PROGRAM IP237
VAR
	
	timer				: TON;
	nState				: INT := STATE_INIT;
	
	fbInit237_01_5500			: FB_InitPM;
	fbInit237_02_5500			: FB_InitPM;
	fbInit237_03_5500			: FB_InitPM;
	fbInit237_04_5500			: FB_InitPM;
	fbInit237_05_5500			: FB_InitPM;
	
	fbRead237_01_5500			: FB_PM_ION_9000;
	fbRead237_02_5500			: FB_PM_ION_9000;
	
	//Update 29-08-2022
	fbRead237_03_5500			: FB_ReadPM5350;
	
	//Update 29-08-2022
	fbRead237_04_5500			: FB_ReadPM5350;
	
	//Update 29-08-2022
	fbRead237_05_5500			: FB_ReadPM5350;
	
	
	ipAddr						: STRING := '10.91.37.237';
	nCount						: DINT;
	nQuantity					: WORD:=125;
	nMBAddr						: WORD:=1;
	bExec						: BOOL;
	bBusy						: BOOL;
	bError						: BOOL;
	nErrorId					:UDINT;
	cbRead						: UDINT;
	bOnTest						:bool;
	PMRawDataTest				:ST_PowerMeter;
	// UPDATE BY SUN
	fbInit237_06_5350			: FB_InitPM;
	fbInit237_07_5350			: FB_InitPM;
	fbInit237_08_5350			: FB_InitPM;
	fbInit237_09_5350			: FB_InitPM;
	fbInit237_10_5350			: FB_InitPM;
	fbInit237_11_5350			: FB_InitPM;
	fbInit237_12_5350			: FB_InitPM;
	fbInit237_13_5350			: FB_InitPM;
	
	fbRead237_06_5350			: FB_ReadPM5350;
	fbRead237_07_5350			: FB_ReadPM5350;
	fbRead237_08_5350			: FB_ReadPM5350;
	fbRead237_09_5350			: FB_ReadPM5350;
	fbRead237_10_5350			: FB_ReadPM5350;
	fbRead237_11_5350			: FB_ReadPM5350;
	fbRead237_12_5350			: FB_ReadPM5350;
	fbRead237_13_5350			: FB_ReadPM5350;
	
END_VAR

VAR CONSTANT
	STATE_INIT			:	INT		:= 0;
	STATE_WAIT_CMD		: 	INT		:= 5;
	STATE_READ1			:	INT		:= 10;
	STATE_READ2			:	INT		:= 20;
	STATE_READ3			:	INT		:= 30;
	STATE_READ4			:	INT		:= 40;
	STATE_READ5			:	INT		:= 50;
	////////////////////////////////////////
	STATE_READ6 		:	INT		:= 60;
	STATE_READ7			:	INT		:= 70;
	STATE_READ8			:	INT		:= 80;
	STATE_READ9			:	INT		:= 90;
	STATE_READ10		:	INT		:= 100;
	STATE_READ11		:	INT		:= 110;
	STATE_READ12		:	INT		:= 120;
	STATE_READ13		:	INT		:= 130;
		

END_VAR

CASE nState OF
	STATE_INIT:
		fbInit237_01_5500(	sIpAddress	:= '10.91.37.227',
							nPort		:= 502,
							nUnitID		:= 255,
							PM			:= pmDev.DB07_01_5500);
		fbInit237_02_5500(	sIpAddress	:= '10.91.37.228',
							nPort		:= 502,
							nUnitID		:= 255,
							PM			:= pmDev.DB07_02_5500);
		fbInit237_03_5500(	sIpAddress	:= '10.91.37.237',
							nPort		:= 502,
							nUnitID		:= 3,
							PM			:= pmDev.DB07_03_5500);
		fbInit237_04_5500(	sIpAddress	:= '10.91.37.237',
							nPort		:= 502,
							nUnitID		:= 4,
							PM			:= pmDev.DB07_04_5500);
		fbInit237_05_5500(	sIpAddress	:= '10.91.37.237',
							nPort		:= 502,
							nUnitID		:= 5,
							PM			:= pmDev.DB07_05_5500);
		// updata by sun///////////////////////////////////////////////
		
		fbInit237_06_5350(	sIpAddress	:= '10.91.37.237',
							nPort		:= 502,
							nUnitID		:= 6,
							PM			:= pmDev.DB07_06_5350);
							
		fbInit237_07_5350(	sIpAddress	:= '10.91.37.237',
							nPort		:= 502,
							nUnitID		:= 7,
							PM			:= pmDev.DB07_07_5350);
							
		fbInit237_08_5350(	sIpAddress	:= '10.91.37.237',
							nPort		:= 502,
							nUnitID		:= 8,
							PM			:= pmDev.DB07_08_5350);
							
		fbInit237_09_5350(	sIpAddress	:= '10.91.37.237',
							nPort		:= 502,
							nUnitID		:= 9,
							PM			:= pmDev.DB07_09_5350);
							
		fbInit237_10_5350(	sIpAddress	:= '10.91.37.237',
							nPort		:= 502,
							nUnitID		:= 10,
							PM			:= pmDev.DB07_10_5350);
							
		fbInit237_11_5350(	sIpAddress	:= '10.91.37.237',
							nPort		:= 502,
							nUnitID		:= 11,
							PM			:= pmDev.DB07_11_5350);
							
		fbInit237_12_5350(	sIpAddress	:= '10.91.37.237',
							nPort		:= 502,
							nUnitID		:= 12,
							PM			:= pmDev.DB07_12_5350);
							
		fbInit237_13_5350(	sIpAddress	:= '10.91.37.237',
							nPort		:= 502,
							nUnitID		:= 13,
							PM			:= pmDev.DB07_13_5350);
							
		timer(In:=TRUE, PT:= TIME_INIT);
		IF timer.Q THEN
			timer(In:=FALSE);
			nState	:= STATE_WAIT_CMD;
		END_IF
			
	STATE_WAIT_CMD:
			;
			
	STATE_READ1:
		fbRead237_01_5500(
			bExecute:=TRUE,
			PM:= pmDev.DB07_01_5500);
		IF NOT fbRead237_01_5500.Q THEN
			nState	:= STATE_READ2;
			fbRead237_01_5500(
				bExecute:=FALSE,
				PM:= pmDev.DB07_01_5500);
		END_IF
		
	STATE_READ2:
		fbRead237_02_5500(
			bExecute:=TRUE,
			PM:= pmDev.DB07_02_5500);
		IF NOT fbRead237_02_5500.Q THEN
			nState	:= STATE_READ3;
			fbRead237_02_5500(
				bExecute:=FALSE,
				PM:= pmDev.DB07_02_5500);
		END_IF	
	
	STATE_READ3:
	
		
		fbRead237_03_5500(
			bExecute:=TRUE,
			PM:= pmDev.DB07_03_5500);
		IF NOT fbRead237_03_5500.Q THEN
			nState	:= STATE_READ4;
			fbRead237_03_5500(
				bExecute:=FALSE,
				PM:= pmDev.DB07_03_5500);
		END_IF	
		
	STATE_READ4:
	
		
		fbRead237_04_5500(
			bExecute:=TRUE,
			PM:= pmDev.DB07_04_5500);
		IF NOT fbRead237_04_5500.Q THEN
			nState	:= STATE_READ5;
			fbRead237_04_5500(
				bExecute:=FALSE,
				PM:= pmDev.DB07_04_5500);
		END_IF
		
	STATE_READ5:
	
	
		fbRead237_05_5500(
			bExecute:=TRUE,
			PM:= pmDev.DB07_05_5500);
		IF NOT fbRead237_05_5500.Q THEN
			nState	:= STATE_READ6;
			fbRead237_05_5500(
				bExecute:=FALSE,
				PM:= pmDev.DB07_05_5500);
		END_IF
	
		////////////////////////////update by Sun
		
	STATE_READ6:
	
		fbRead237_06_5350(
			bExecute:=TRUE,
			PM:= pmDev.DB07_06_5350);
		IF NOT fbRead237_06_5350.Q THEN
			nState	:= STATE_READ7;
			fbRead237_06_5350(
				bExecute:=FALSE,
				PM:= pmDev.DB07_06_5350);
		END_IF
	
	STATE_READ7:
	
		fbRead237_07_5350(
			bExecute:=TRUE,
			PM:= pmDev.DB07_07_5350);
		IF NOT fbRead237_07_5350.Q THEN
			nState	:= STATE_READ8;
			fbRead237_07_5350(
				bExecute:=FALSE,
				PM:= pmDev.DB07_07_5350);
		END_IF
	
	STATE_READ8:
	
		fbRead237_08_5350(
			bExecute:=TRUE,
			PM:= pmDev.DB07_08_5350);
		IF NOT fbRead237_08_5350.Q THEN
			nState	:= STATE_READ9;
			fbRead237_08_5350(
				bExecute:=FALSE,
				PM:= pmDev.DB07_08_5350);
		END_IF
	
	STATE_READ9:
	
		fbRead237_09_5350(
			bExecute:=TRUE,
			PM:= pmDev.DB07_09_5350);
		IF NOT fbRead237_09_5350.Q THEN
			nState	:= STATE_READ10;
			fbRead237_09_5350(
				bExecute:=FALSE,
				PM:= pmDev.DB07_09_5350);
		END_IF
		
	STATE_READ10:
	
		fbRead237_10_5350(
			bExecute:=TRUE,
			PM:= pmDev.DB07_10_5350);
		IF NOT fbRead237_10_5350.Q THEN
			nState	:= STATE_READ11;
			fbRead237_10_5350(
				bExecute:=FALSE,
				PM:= pmDev.DB07_10_5350);
		END_IF
	
	STATE_READ11:
	
		fbRead237_11_5350(
			bExecute:=TRUE,
			PM:= pmDev.DB07_11_5350);
		IF NOT fbRead237_11_5350.Q THEN
			nState	:= STATE_READ12;
			fbRead237_11_5350(
				bExecute:=FALSE,
				PM:= pmDev.DB07_11_5350);
		END_IF
	
	STATE_READ12:
	
		fbRead237_12_5350(
			bExecute:=TRUE,
			PM:= pmDev.DB07_12_5350);
		IF NOT fbRead237_12_5350.Q THEN
			nState	:= STATE_READ13;
			fbRead237_12_5350(
				bExecute:=FALSE,
				PM:= pmDev.DB07_12_5350);
		END_IF
	
	STATE_READ13:
	
		fbRead237_13_5350(
			bExecute:=TRUE,
			PM:= pmDev.DB07_13_5350);
		IF NOT fbRead237_13_5350.Q THEN
			nState	:= STATE_WAIT_CMD;
			fbRead237_13_5350(
				bExecute:=FALSE,
				PM:= pmDev.DB07_13_5350);
		END_IF
	

	
END_CASE

PROPERTY Busy : Bool
GET
Busy := nState <> STATE_WAIT_CMD;
END_GET
END_PROPERTY

METHOD Mr_Read : BOOL
VAR_INPUT
END_VAR
IF nState = STATE_WAIT_CMD THEN
	nState := STATE_READ1;
END_IF
END_METHOD

END_PROGRAM

(* stored: Version 1.1.0.1, ProductVersion 3.1.4024.12
   POU IP237: Id {2f627f47-e9b3-4a94-9dbe-15db80907e0e}, SpecialFunc None
   Property Busy: Id {6abd9ec0-03cd-4794-9f62-392a343c627e}
   Get Get: Id {b236e423-d81a-4f42-90f0-9b04694f89f7}
   Method Mr_Read: Id {5c83eeeb-4f9e-4abc-a1cd-ed0ee1db8d68} *)
